TYPE MultiAxis_monitor_typ :
STRUCT
END_STRUCT
END_TYPE

(* stored: Version 1.1.0.1, ProductVersion 3.1.4024.3
   DUT MultiAxis_monitor_typ: Id {cacc8cc8-0646-0fe8-3a23-1d9423cbc9f3} *)
